TEXTLIST ModeStates
  0 = 'No State'
  1 = 'Power Off'
  2 = 'Power On'
  3 = 'Manual Mode'
  4 = 'Auto Mode'
  5 = 'Auto Cycling'
  6 = 'Semi Auto'
  7 = 'Fault'
  8 = 'Bypass'
  9 = 'Auto Cycle Stopping'
  10 = 'State2'
   = ''
END_TEXTLIST

(* stored: Version 1.1.0.1, ProductVersion 3.1.4024.12
   TextList ModeStates: Id {9ed31934-f9ea-44f4-865f-53c4c08ab203} *)
